// TIA Portal project "MES-tracing-bullet" (V15.1)

(* hardware
DEVICE "S7-1200 station_1"  S7-1200 Station
   slot 0: "Rack_0"  S7-1200 Rack  Rack  V1.0
   slot 1: "PLC_1"  CPU 1214C DC/DC/DC  6ES7 214-1AG40-0XB0  V4.0
*)

// ===== PLC "PLC_1"  CPU 1214C DC/DC/DC =====

// folder: PLCUT

TYPE "PLCUT"
   STRUCT
      pc : "PLCUT-PC";
      plc : "PLCUT-PLC";
   END_STRUCT;
END_TYPE

TYPE "PLCUT-PC"
   STRUCT
      execute : Bool;
      ts_index : Int;
      tc_index : Int;
   END_STRUCT;
END_TYPE

TYPE "PLCUT-PLC"
   STRUCT
      valid : Bool;
      processed : Bool;
      result : Bool;
      ts_name : String[128];
      tc_name : String[128];
   END_STRUCT;
END_TYPE

// folder: mes

TYPE "mes-struct-1"
   STRUCT
      LiveCheck : Byte;
      JIT_status : Byte;
      PLC_status : Byte;
      JobNr : Array[0..9] of Char;
      CallOffDateTime : Array[0..15] of Char;
      VehicleNo : Array[0..12] of Char;
      RearWindowType : String[18];
      Model : Byte;
   END_STRUCT;
END_TYPE

TYPE "mes-struct-2"
   STRUCT
      LiveCheck : Byte;
      JIT_status : Byte;
      PLC_status : Byte;
      JobNr : Array[0..9] of Char;
      VehicleNo : Array[0..12] of Char;
      RearWindowType : String[18];
   END_STRUCT;
END_TYPE

TYPE "mes-struct-3"
   STRUCT
      LiveCheck : Byte;
      JIT_status : Byte;
      PLC_status : Byte;
      JobNr : Array[0..9] of Char;
      VehicleNo : Array[0..12] of Char;
      RearWindowType : String[18];
      GlassID : Array[0..9] of Char;
      flag4 : Bool;
   END_STRUCT;
END_TYPE

// folder: (top level)

DATA_BLOCK "MES-1"   // DB1
{ S7_Optimized_Access := 'FALSE' }
VERSION : 0.1
   VAR
      self : "mes-struct-1";
   END_VAR
BEGIN
END_DATA_BLOCK

DATA_BLOCK "MES-2"   // DB2
{ S7_Optimized_Access := 'FALSE' }
VERSION : 0.1
   VAR
      self : "mes-struct-2";
   END_VAR
BEGIN
END_DATA_BLOCK

DATA_BLOCK "MES-3"   // DB3
{ S7_Optimized_Access := 'FALSE' }
VERSION : 0.1
   VAR
      self : "mes-struct-3";
   END_VAR
BEGIN
END_DATA_BLOCK

// folder: PLCUT

DATA_BLOCK "DB_PLCUT"   // DB4
{ S7_Optimized_Access := 'FALSE' }
VERSION : 0.1
   VAR
      self : "PLCUT";
   END_VAR
BEGIN
END_DATA_BLOCK

// folder: (top level)

ORGANIZATION_BLOCK "Main"   // OB1, LAD, ProgramCycle
TITLE = "Main Program Sweep (Cycle)"
{ S7_Optimized_Access := 'TRUE' }
VERSION : 0.1
   VAR_INPUT
      Initial_Call : Bool;   // Initial call of this OB
      Remanence : Bool;   // =True, if remanent data are available
   END_VAR
BEGIN

REGION Network 1
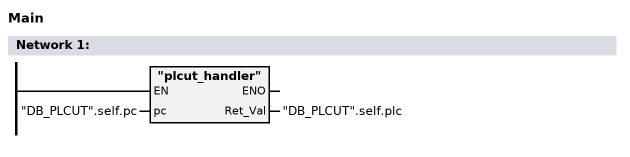
   RUNG wire#powerrail
      "plcut_handler"(pc := "DB_PLCUT".self.pc, Ret_Val => "DB_PLCUT".self.plc)
   END_RUNG
   // the same network as SCL:
   "DB_PLCUT".self.plc := "plcut_handler"(pc := "DB_PLCUT".self.pc);
END_REGION
END_ORGANIZATION_BLOCK

// folder: PLCUT

FUNCTION "plcut_handler" : "PLCUT-PLC"   // FC1, SCL
{ S7_Optimized_Access := 'TRUE' }
VERSION : 0.1
   VAR_INPUT
      pc : "PLCUT-PC";
   END_VAR
BEGIN
   IF #pc.execute = TRUE
   THEN
       IF #pc.ts_index = 0
       THEN
           #plcut_handler := "test_suite_1"(tc_index := #pc.tc_index, ts_name := 'test suite 1');
       ELSE
           #plcut_handler := "plcut_invalid"();
       END_IF;
   ELSE
       #plcut_handler := "plcut_nil"();
   END_IF;
END_FUNCTION

// folder: PLCUT/TS/TS-1

FUNCTION "test_suite_1" : "PLCUT-PLC"   // FC2, SCL
{ S7_Optimized_Access := 'TRUE' }
VERSION : 0.1
   VAR_INPUT
      tc_index : Int;
      ts_name : String;
   END_VAR
BEGIN

   IF #tc_index = 0
   THEN
       #test_suite_1 := "plcut_assert"(evaluation := true, ts_name:=#ts_name, tc_name := 'assert test 1');
   ELSIF #tc_index = 1
   THEN
       #test_suite_1 := "plcut_assert"(evaluation := true, ts_name := #ts_name, tc_name := 'assert test 2');
   ELSE
       #test_suite_1 := "plcut_invalid"();
   END_IF;
END_FUNCTION

// folder: PLCUT/api

FUNCTION "plcut_nil" : "PLCUT-PLC"   // FC3, SCL
{ S7_Optimized_Access := 'TRUE' }
VERSION : 0.1
   VAR_TEMP
      nil : "PLCUT-PLC";
   END_VAR
BEGIN
   #plcut_nil := #nil;
END_FUNCTION

FUNCTION "plcut_invalid" : "PLCUT-PLC"   // FC4, SCL
{ S7_Optimized_Access := 'TRUE' }
VERSION : 0.1
   VAR_TEMP
      nil : "PLCUT-PLC";
   END_VAR
BEGIN

   #nil := "plcut_nil"();
   #nil.processed := true;

   #plcut_invalid := #nil;
END_FUNCTION

FUNCTION "plcut_assert" : "PLCUT-PLC"   // FC5, SCL
{ S7_Optimized_Access := 'TRUE' }
VERSION : 0.1
   VAR_INPUT
      evaluation : Bool;
      ts_name : String;
      tc_name : String;
   END_VAR
   VAR_TEMP
      assert : "PLCUT-PLC";
   END_VAR
BEGIN

   #assert.valid := true;
   #assert.processed := true;
   #assert.result := #evaluation;
   #assert.tc_name := #tc_name;
   #assert.ts_name := #ts_name;

   #plcut_assert := #assert;
END_FUNCTION